// TIA Portal V17 export
// export: Created 2022-06-27T13:58:35.9641236Z, ExportSetting WithDefaults, DisplayName Totally Integrated Automation Portal, DisplayVersion V17 Update 3, DisplayName TIA Portal Openness, DisplayVersion V17 Update 3, DisplayName TIA Portal Version Control Interface, DisplayVersion V17, DisplayName SINAMICS Startdrive Advanced, DisplayVersion V17 Update1, DisplayName SINAMICS Startdrive G110M, G120, G120C, G120D, G120P, G115D, DisplayVersion V17 Update1, DisplayName SINAMICS Startdrive G130, G150, S120, S150, SINAMICS MV, S210, DisplayVersion V17 Update1, DisplayName STEP 7 Professional, DisplayVersion V17 Update 3, DisplayName STEP 7 Safety, DisplayVersion V17, DisplayName WinCC UA Professional, DisplayVersion V17 Update 3
FUNCTION_BLOCK "S061_DIGITAL_INPUTS"   // FB61, LAD
{ S7_Optimized_Access := 'TRUE' }
VERSION : 0.1
// stored: AutoNumber false, IsIECCheckEnabled false, IsRetainMemResEnabled false, MemoryReserve 100, SetENOAutomatically false, UDAEnableTagReadback false
BEGIN

REGION Network 1: U33-2D - Burner Fan On
END_REGION

REGION Network 2: U35-2D - Roasting Chamber 1 Motor On
END_REGION

REGION Network 3: U35-4D - Roasting Chamber 2 Motor On
END_REGION

REGION Network 4: U37-2D - Cooler Chamber 1 Motor On
END_REGION

REGION Network 5: U37-3D - Cooler Chamber 2 Motor On
END_REGION

REGION Network 6: K98-4E - Burner Damaged
END_REGION

REGION Network 7: K98-6E - Bruner On
END_REGION

REGION Network 8: K98-3E - Burner Combuster On
END_REGION

REGION Network 9: K43-2D - Energy Fault
END_REGION

REGION Network 10: KSV44-5C - Safety Relay On
END_REGION

REGION Network 11: FCI - Internal Voltage Source OK
END_REGION

REGION Network 12: FCE - External Voltage Source OK
END_REGION

REGION Network 13: KSV46-4C - Chamber 1 Safety Relay On
END_REGION

REGION Network 14: KSV46-8C - Chamber 2 Safety Relay On
END_REGION

REGION Network 15: KSV47-4C - Cooling Chamber 1 Safety Relay On
END_REGION

REGION Network 16: KSV47-8C - Cooling Chamber 2 Safety Relay On
END_REGION

REGION Network 17: TCTL - Coffee Transportation Turned On
END_REGION

REGION Network 18: ZSV46-2C - Chamber 1 Manual Override Safety Limit Switch
END_REGION

REGION Network 19: ZSV46-6C - Chamber 2 Manual Override Safety Limit Switch
END_REGION

REGION Network 20: ZSV47-2C - Cooler 1 Manual Override Safety Limit Switch
END_REGION

REGION Network 21: ZSV47-6C - Cooler 2 Manual Override Safety Limit Switch
END_REGION

REGION Network 22: G43-4C-1 - Nobreak Low Battery Status
END_REGION

REGION Network 23: G43-4C-2 - Nobreak Network Status
END_REGION

REGION Network 24: LSL66-2C - Level Sensor "catador"
END_REGION

REGION Network 25: ZSL66-4B - Chamber 1 Intake Open Limit Switch
END_REGION

REGION Network 26: ZSH66-5B - Chamber 1 Intake Close Limit Switch
END_REGION

REGION Network 27: ZSL66-6B - Chamber 1 Discharge Open Limit Switch
END_REGION

REGION Network 28: ZSH66-7B - Chamber 1 Discharge Close Limit Switch
END_REGION

REGION Network 29: ZSL66-8B - Cooler 1 Discharge Close Limit Switch
END_REGION

REGION Network 30: ZSH66-9B - Cooler 1 Discharge Open Limit Switch
END_REGION

REGION Network 31: ZSL67-2B - Chamber 2 Intake Close Limit Switch
END_REGION

REGION Network 32: ZSH67-3B - Chamber 2 Intake Open Limit Switch
END_REGION

REGION Network 33: ZSL67-4B - Chamber 2 Discharge Close Limit Switch
END_REGION

REGION Network 34: ZSH67-5B - Chamber 2 Discharge Open Limit Switch
END_REGION

REGION Network 35: ZSL67-6B - Cooler 2 Discharge Open Limit Switch
END_REGION

REGION Network 36: ZSH67-7B - Cooler 2 Discharge Close Limit Switch
END_REGION

REGION Network 37: ZSL67-8B - Chamber 2 Roaster Fan Limit Switch
END_REGION

REGION Network 38: ZSH67-9B - Chamber 1 Roaster Fan Limit Switch
END_REGION

REGION Network 39: ZSL68-2B - Chamber 2 Dryer Fan Limit Switch
END_REGION

REGION Network 40: ZSH68-3B - Chamber 1 Dryer Fan Limit Switch
END_REGION

REGION Network 41: ZSL68-4B - Chamber 1 Cooler Fan Limit Switch
END_REGION

REGION Network 42: ZSH68-5B - Chamber 2 Cooler Fan Limit Switch
END_REGION

REGION Network 43: ZSL68-6B - Branch Valve Manual Bagging Direction
END_REGION

REGION Network 44: ZSH68-7B - Branch Valve Transport Direction
END_REGION

REGION Network 45: ZSL68-8B - Branch Valve Elevator Direction
END_REGION

REGION Network 46: ZSH68-9B - Branch Valve Air Conveyor Direction
END_REGION

REGION Network 47: LSH69-2B - Chamber 1 Raw Coffee Silo Level 1 Capacitive Sensor
END_REGION

REGION Network 48: LSL69-3B - Chamber 1 Raw Coffee Silo Level 2 Capacitive Sensor
END_REGION

REGION Network 49: LSH69-5B - Chamber 2 Raw Coffee Silo Level 1 Capacitive Sensor
END_REGION

REGION Network 50: LSL69-6B - Chamber 2 Raw Coffee Silo Level 2 Capacitive Sensor
END_REGION

REGION Network 51: SSL69-8B - Chamber 1 Rotation Sensor
END_REGION

REGION Network 52: SSL69-9B - Chamber 2 Rotation Sensor
END_REGION

REGION Network 53: SSL70-2B - Cooler 1 Rotation Sensor
END_REGION

REGION Network 54: SSL70-3B - Cooler 2 Rotation Sensor
END_REGION

REGION Network 55: SSL70-4B - Cooler Conveyor Rotation Sensor
END_REGION

REGION Network 56: SSL70-5B - Tilted Conveyor Rotation Sensor
END_REGION

REGION Network 57: LSL70-6B - Water Reservoir Level Sensor
END_REGION

REGION Network 58: LSL70-7B - Cooler Bucket 1 Capacitive Sensor
END_REGION

REGION Network 59: LSL70-8B - Cooler Bucket 1 Capacitive Sensor
END_REGION

REGION Network 60: PSL70-9B - Preassured Air Gauge
END_REGION

REGION Network 61: HR71-2BA - Water Pump Intake Manual Valve Open
END_REGION

REGION Network 62: HR71-2BF - Water Pump Intake Manual Valve Close
END_REGION

REGION Network 63: ZSL71-4B - Limit Switch Cyclones Conveyor
END_REGION

REGION Network 64: ZSL71-5B - Limit Switch Tilted Conveyor
END_REGION

REGION Network 65: ZSH71-5B - Chamber 1 Hot Air Pneumatic Actuator Open
END_REGION

REGION Network 66: ZSL71-7B - Chamber 1 Hot Air Pneumatic Actuator Close
END_REGION

REGION Network 67: ZSH71-8B - Chamber 2 Hot Air Pneumatic Actuator Open
END_REGION

REGION Network 68: ZSL71-9B - Chamber 2 Hot Air Pneumatic Actuator Close
END_REGION

REGION Network 69: ZSH72-2B - Chamber 1 Ambient Air Pneumatic Actuator Open
END_REGION

REGION Network 70: ZSL72-3B - Chamber 1 Ambient Air Pneumatic Actuator Close
END_REGION

REGION Network 71: ZSH72-4B - Chamber 2 Ambient Air Pneumatic Actuator Open
END_REGION

REGION Network 72: ZSL72-5B - Chamber 2 Ambient Air Pneumatic Actuator Close
END_REGION

REGION Network 73: SSL72-6B - Roaster Cyclone Rotary Valve Rotation Sensor
END_REGION

REGION Network 74: SSL72-7B - Roaster Fan Rotation Sensor
END_REGION

REGION Network 75: SSL72-8B - Dryer Fan Rotation Sensor
END_REGION

REGION Network 76: PSL72-9B - Cooler Fan Rotation Sensor
END_REGION

REGION Network 77: S73-2B - Manual Bagging Key
END_REGION

REGION Network 78: S73-3B - Automatic Bagging Key
END_REGION

REGION Network 79: PSL73-4B - Chamber 1 Ambient Air Fan Preassure Gauge
END_REGION

REGION Network 80: PSL73-5B - Chamber 2 Ambient Air Fan Preassure Gauge
END_REGION

REGION Network 81: SSL73-6B - Cooler Cyclone Rotary Valve Rotation Sensor
END_REGION

REGION Network 82: SSL73-7B - Dryer 1 Cyclone Rotary Valve Rotation Sensor
END_REGION

REGION Network 83: SSL73-8B - Dryer 2 Cyclone Rotary Valve Rotation Sensor
END_REGION

REGION Network 84: SSL73-9B - Cyclones Conveyor Rotation Sensor
END_REGION

REGION Network 85: HSH74-2B - Manual Valve Air Intake
END_REGION

REGION Network 86: HSL74-3B - Chamber 1 Water Injection Manual Valve Closed
END_REGION

REGION Network 87: HSL74-4B - Chamber 2 Water Injection Manual Valve Closed
END_REGION

REGION Network 88: HSL74-5B - Cooler 1 Water Injection Manual Valve Closed
END_REGION

REGION Network 89: HSL74-6B - Cooler 2 Water Injection Manual Valve Closed
END_REGION

REGION Network 90: HSL74-7B - Air Reservoir Relief Manual Valve Closed
END_REGION

REGION Network 91: HSL74-8B - Water Reservoir Air Relief Manual Valve Closed
END_REGION

REGION Network 92: HSH74-9B - Roaster Water Intake After Pump Manual Valve Opened
END_REGION

REGION Network 93: HSH75-2B - Roaster Water Intake Manual Valve Opened
END_REGION

REGION Network 94: HSH75-3B - Pump Water Manual Valve Opened
END_REGION

REGION Network 95: PSL75-4B - Water Flow Rate
END_REGION

REGION Network 96: FSL75-5B - Air Intake Preassure Gauge
END_REGION

REGION Network 97: ZSL75-6B - Cooler Conveyor Limit Switch
END_REGION

REGION Network 98: K94-4D - Gas Flow Rate
END_REGION

REGION Network 99: K94-7D - Oil Flow Rate
END_REGION
END_FUNCTION_BLOCK
